FUNCTION_BLOCK FB_Cylinder_DualSensor EXTENDS FB_CylinderBase
VAR_INPUT
END_VAR
VAR_OUTPUT
END_VAR
VAR
	fbSensor_Extended							: FB_Sensor;
	fbSensor_Retracted							: FB_Sensor;
END_VAR

METHOD HardwareUpdate : BOOL
VAR_INPUT
END_VAR
fbSensor_Extended.CyclicLogic();
fbSensor_Retracted.CyclicLogic();

bExtendedFeedback:= fbSensor_Extended.Active;
bRetractedFeedback := fbSensor_Retracted.Active;
END_METHOD

END_FUNCTION_BLOCK

(* stored: Version 1.1.0.1, ProductVersion 3.1.4024.9
   POU FB_Cylinder_DualSensor: Id {548cb264-8e0d-49f7-a008-32e71d85168c}, SpecialFunc None
   Folder 01_SUPER_Overrides: Id {4dc883f4-4cfb-47b5-86e5-2bb7b1d9b438}
   Method HardwareUpdate: Id {692e3844-c464-4955-a750-d8f7a26ca635} *)
